(* IEC 61131-3 sources: SIMERLIFT/logiwork_simerlift_80v/logiwork_simerlift_80v/HEMAbattery/src_FBD/fbdCommon, 9 files *)

(* ---- fMaxSint.iecst ---- *)
FUNCTION fMaxSint  {
    width := 200;
  }

VAR_INPUT
	arr:ARRAY[0..15] OF SINT;
	sizeof:USINT;
END_VAR

VAR_OUTPUT
	max : SINT;
END_VAR

VAR
i:USINT;

END_VAR

max:=-128;

FOR i:=1 TO sizeof By 1 DO
	IF max<arr[i-1] THEN
		max:=arr[i-1];
	END_IF;
END_FOR;

END_FUNCTION

(* ---- fMinUint.iecst ---- *)
FUNCTION fMinUint  {
    width := 200;
  }

VAR_INPUT
	arr:ARRAY[0..15] OF UINT;
	sizeof:USINT;
END_VAR

VAR_OUTPUT
	min : UINT;
END_VAR

VAR
i:USINT;

END_VAR

min:=16#FFFF;

FOR i:=1 TO sizeof By 1 DO
	IF min>arr[i-1] THEN
		min:=arr[i-1];
	END_IF;
END_FOR;

END_FUNCTION

(* ---- RBIT.iecfbd ---- *)
FUNCTION RBIT
  VAR_INPUT
    start : INT;
    len : INT;
    INbit : LWORD;
  END_VAR
  VAR_OUTPUT
    OUTbit : LWORD;
  END_VAR

  (*

    // Network 1:
    SHR(IN := INbit, N := start, SHR => @C(12).SHR);
    SUB(IN1 := 64, IN2 := len, SUB => @C(2).SUB);
    SHR(IN := 16#FFFFFFFFFFFFFFFF, N := @C(2).SUB, SHR => @C(6).SHR);
    AND(IN1 := @C(12).SHR, IN2 := @C(6).SHR, AND => OUTbit);

  *)

  @VF(1) : @E(64), @R(460.0, 160.0, 80.0, 19.0), INT;
  @C(2) : @F(SUB), @R(590.0, 160.0, 40.0, 38.0), INT, @I(@N(IN1), @L(9.5)), @I(@N(IN2), @L(29.5)), @O(@N(SUB), @R(9.5));
  @VF(3) : @E(len), @R(230.0, 180.0, 140.0, 19.0);
  @C(6) : @F(SHR), @R(670.0, 140.0, 100.0, 38.0), LWORD, @I(@N(IN), @L(9.5)), @I(@N(N), @L(29.5)), @O(@N(SHR), @R(9.5));
  @VF(8) : @E(16#FFFFFFFFFFFFFFFF), @R(460.0, 140.0, 170.0, 19.0), LWORD;
  @VF(10) : @E(INbit), @R(230.0, 100.0, 140.0, 19.0);
  @VF(11) : @E(start), @R(230.0, 120.0, 140.0, 19.0);
  @C(12) : @F(SHR), @R(670.0, 100.0, 100.0, 38.0), LWORD, @I(@N(IN), @L(9.5)), @I(@N(N), @L(29.5)), @O(@N(SHR), @R(9.5));
  @C(15) : @F(AND), @R(830.0, 100.0, 40.0, 38.0), LWORD, @I(@N(IN1), @L(9.5)), @I(@N(IN2), @L(29.5)), @O(@N(AND), @R(9.5));
  @VF(18) : @E(OUTbit), @R(1000.0, 100.0, 140.0, 19.0);

  @G(4) :
     @L(@VF(3).o, @C(2).IN2)
    ;
  @G(5) :
     @L(@VF(1).o, @C(2).IN1)
    ;
  @G(7) :
     @L(@C(2).SUB, @C(6).N)
    ;
  @G(9) :
     @L(@VF(8).o, @C(6).IN)
    ;
  @G(13) :
     @L(@VF(10).o, @C(12).IN)
    ;
  @G(14) :
     @L(@VF(11).o, @C(12).N)
    ;
  @G(16) :
     @L(@C(12).SHR, @C(15).IN1)
    ;
  @G(17) :
     @L(@C(6).SHR, @C(15).IN2)
    ;
  @G(19) :
     @L(@C(15).AND, @VF(18).i)
    ;
END_FUNCTION

(* ---- WFLT.iecfbd ---- *)
FUNCTION WFLT
  VAR_INPUT
    start : INT;
    len : INT;
    prm : LREAL;
    ofs : LREAL;
    res : LREAL;
  END_VAR
  VAR_OUTPUT
    OUTbit : LWORD;
  END_VAR

  (*

    // Network 1:
    SHL(IN := 16#FFFFFFFFFFFFFFFF, N := start, SHL => @C(4).SHL);
    ADD(IN1 := start, IN2 := len, ADD => @C(7).ADD);
    SUB(IN1 := 64, IN2 := @C(7).ADD, SUB => @C(12).SUB);
    SHR(IN := 16#FFFFFFFFFFFFFFFF, N := @C(12).SUB, SHR => @C(15).SHR);
    AND(IN1 := @C(4).SHL, IN2 := @C(15).SHR, AND => @C(19).AND);
    SUB(IN1 := prm, IN2 := ofs, SUB => @C(29).SUB);
    DIV(IN1 := @C(29).SUB, IN2 := res, DIV => @C(32).DIV);
    TO_LWORD(IN := @C(32).DIV, TO_LWORD => @C(36).TO_LWORD);
    SHL(IN := @C(36).TO_LWORD, N := start, SHL => @C(23).SHL);
    AND(IN1 := @C(19).AND, IN2 := @C(23).SHL, AND => OUTbit);

  *)

  @C(4) : @F(SHL), @R(670.0, 80.0, 100.0, 38.0), LWORD, @I(@N(IN), @L(9.5)), @I(@N(N), @L(29.5)), @O(@N(SHL), @R(9.5));
  @C(12) : @F(SUB), @R(930.0, 100.0, 40.0, 38.0), INT, @I(@N(IN1), @L(9.5)), @I(@N(IN2), @L(29.5)), @O(@N(SUB), @R(9.5));
  @C(15) : @F(SHR), @R(1030.0, 80.0, 100.0, 38.0), LWORD, @I(@N(IN), @L(9.5)), @I(@N(N), @L(29.5)), @O(@N(SHR), @R(9.5));
  @C(19) : @F(AND), @R(1190.0, 60.0, 40.0, 38.0), LWORD, @I(@N(IN1), @L(9.5)), @I(@N(IN2), @L(29.5)), @O(@N(AND), @R(9.5));
  @C(7) : @F(ADD), @R(670.0, 120.0, 40.0, 38.0), INT, @I(@N(IN1), @L(9.5)), @I(@N(IN2), @L(29.5)), @O(@N(ADD), @R(9.5));
  @C(22) : @F(AND), @R(1320.0, 140.0, 40.0, 38.0), LWORD, @I(@N(IN1), @L(9.5)), @I(@N(IN2), @L(29.5)), @O(@N(AND), @R(9.5));
  @C(23) : @F(SHL), @R(670.0, 160.0, 100.0, 38.0), LWORD, @I(@N(IN), @L(9.5)), @I(@N(N), @L(29.5)), @O(@N(SHL), @R(9.5));
  @VF(8) : @E(16#FFFFFFFFFFFFFFFF), @R(470.0, 80.0, 170.0, 19.0), LWORD;
  @VF(1) : @E(start), @R(130.0, 100.0, 140.0, 19.0);
  @VF(11) : @E(64), @R(820.0, 100.0, 70.0, 19.0), INT;
  @VF(17) : @E(16#FFFFFFFFFFFFFFFF), @R(810.0, 80.0, 170.0, 19.0), LWORD;
  @VF(2) : @E(len), @R(130.0, 140.0, 140.0, 19.0);
  @VF(27) : @E(OUTbit), @R(1400.0, 140.0, 140.0, 19.0);
  @VF(3) : @E(prm), @R(130.0, 160.0, 140.0, 19.0);
  @VF(24) : @E(ofs), @R(130.0, 180.0, 140.0, 19.0);
  @C(29) : @F(SUB), @R(320.0, 160.0, 40.0, 38.0), LREAL, @I(@N(IN1), @L(9.5)), @I(@N(IN2), @L(29.5)), @O(@N(SUB), @R(9.5));
  @C(32) : @F(DIV), @R(400.0, 160.0, 40.0, 38.0), LREAL, @I(@N(IN1), @L(9.5)), @I(@N(IN2), @L(29.5)), @O(@N(DIV), @R(9.5));
  @VF(34) : @E(res), @R(130.0, 200.0, 140.0, 19.0);
  @C(36) : @F(TO_LWORD), @R(460.0, 160.0, 120.0, 18.0), LREAL, @I(@N(IN), @L(9.5)), @O(@N(TO_LWORD), @R(9.5));
  @CP(10) : 609.5, 109.5;

  @G(5) :
     @L(@VF(8).o, @C(4).IN)
    ;
  @G(6) :
     @L(@VF(1).o, @CP(10)),
     @L(@CP(10), @C(4).N),
     @L(@CP(10), @C(7).IN1),
     @L(@CP(10), @C(23).N)
    ;
  @G(13) :
     @L(@VF(11).o, @C(12).IN1)
    ;
  @G(14) :
     @L(@C(7).ADD, @C(12).IN2)
    ;
  @G(16) :
     @L(@C(12).SUB, @C(15).N)
    ;
  @G(18) :
     @L(@VF(17).o, @C(15).IN)
    ;
  @G(9) :
     @L(@VF(2).o, @C(7).IN2)
    ;
  @G(20) :
     @L(@C(15).SHR, @C(19).IN2)
    ;
  @G(21) :
     @L(@C(4).SHL, @C(19).IN1)
    ;
  @G(25) :
     @L(@C(19).AND, @C(22).IN1)
    ;
  @G(26) :
     @L(@C(23).SHL, @C(22).IN2)
    ;
  @G(28) :
     @L(@C(22).AND, @VF(27).i)
    ;
  @G(30) :
     @L(@VF(3).o, @C(29).IN1)
    ;
  @G(31) :
     @L(@VF(24).o, @C(29).IN2)
    ;
  @G(33) :
     @L(@C(29).SUB, @C(32).IN1)
    ;
  @G(35) :
     @L(@VF(34).o, @C(32).IN2)
    ;
  @G(37) :
     @L(@C(32).DIV, @C(36).IN)
    ;
  @G(38) :
     @L(@C(36).TO_LWORD, @C(23).IN)
    ;
END_FUNCTION

(* ---- AVG.iecfbd ---- *)
FUNCTION_BLOCK AVG
  {
    In {index := 0};
    Out {index := 0};
    width := 100;
    height := 18;
  }

  VAR
    Out_Buff : LREAL := 0;
  END_VAR
  VAR_INPUT
    In : LREAL := 0;
  END_VAR
  VAR_OUTPUT
    Out : LREAL := 0;
  END_VAR

  (*

    // Network 1:
    MUL(IN1 := In, IN2 := 0.001, MUL => @C(4).MUL);
    MUL(IN1 := Out_Buff, IN2 := 0.999, MUL => @C(9).MUL);
    ADD(IN1 := @C(4).MUL, IN2 := @C(9).MUL, ADD => (Out, Out_Buff));

  *)

  @VF(1) : @E(In), @R(20.0, 20.0, 220.0, 19.0);
  @VF(2) : @E(Out), @R(520.0, 20.0, 220.0, 19.0);
  @VF(186) : @E(0.001), @R(130.0, 40.0, 110.0, 19.0), LREAL;
  @C(6) : @F(ADD), @R(400.0, 20.0, 40.0, 38.0), LREAL, @I(@N(IN1), @L(9.5)), @I(@N(IN2), @L(29.5)), @O(@N(ADD), @R(9.5));
  @VF(10) : @E(0.999), @R(130.0, 80.0, 110.0, 19.0), LREAL;
  @C(4) : @F(MUL), @R(280.0, 20.0, 40.0, 38.0), LREAL, @I(@N(IN1), @L(9.5)), @I(@N(IN2), @L(29.5)), @O(@N(MUL), @R(9.5));
  @C(9) : @F(MUL), @R(280.0, 60.0, 40.0, 38.0), LREAL, @I(@N(IN1), @L(9.5)), @I(@N(IN2), @L(29.5)), @O(@N(MUL), @R(9.5));
  @VF(12) : @E(Out_Buff), @R(520.0, 40.0, 220.0, 19.0);
  @VF(15) : @E(Out_Buff), @R(20.0, 60.0, 220.0, 19.0);
  @CP(13) : 489.5, 29.5;

  @G(14) :
     @L(@C(6).ADD, @CP(13)),
     @L(@CP(13), @VF(2).i),
     @L(@CP(13), @VF(12).i)
    ;
  @G(5) :
     @L(@VF(1).o, @C(4).IN1)
    ;
  @G(8) :
     @L(@VF(186).o, @C(4).IN2)
    ;
  @G(11) :
     @L(@VF(10).o, @C(9).IN2)
    ;
  @G(3) :
     @L(@C(4).MUL, @C(6).IN1)
    ;
  @G(7) :
     @L(@C(9).MUL, @C(6).IN2)
    ;
  @G(16) :
     @L(@VF(15).o, @C(9).IN1)
    ;
END_FUNCTION_BLOCK

(* ---- CounTim.iecfbd ---- *)
FUNCTION_BLOCK CounTim
  {
    ACCper {index := 2};
    DECper {index := 3};
    PV {index := 4};
    CV {index := 4};
    height := 98;
    width := 210;
    bgColor := "darkseagreen";
  }

  VAR
    FLASH7 : FLASH;
    FLASH8 : FLASH;
    CTUD3 : CTUD;
  END_VAR
  VAR_INPUT
    ACCper : TIME;
    DECper : TIME;
    CU : BOOL;
    CD : BOOL;
    PV : INT;
  END_VAR
  VAR_OUTPUT
    CV : INT;
    QU : BOOL;
    QD : BOOL;
  END_VAR

  (*

    // Network 1:
    AND(IN1 := NOT CTUD3.QU, IN2 := CU, AND => @C(66).AND);
    FLASH7(IN := @C(66).AND, PER := ACCper);
    AND(IN1 := CD, IN2 := NOT CTUD3.QD, AND => @C(68).AND);
    FLASH8(IN := @C(68).AND, PER := DECper);
    CTUD3(CU := FLASH7.OUT, CD := FLASH8.OUT, PV := PV, QU => QU, QD => QD, CV => CV);

  *)

  @C(66) : @F(AND), @R(410.0, 240.0, 40.0, 38.0), BOOL, @I(@N(IN1), @L(9.5), @NEG), @I(@N(IN2), @L(29.5)), @O(@N(AND), @R(9.5));
  @C(39) : @FB(FLASH7), @R(550.0, 260.0, 120.0, 38.0), @I(@N(IN), @L(9.5)), @I(@N(PER), @L(29.5)), @O(@N(OUT), @R(9.5));
  @C(40) : @FB(FLASH8), @R(550.0, 300.0, 120.0, 38.0), @I(@N(IN), @L(9.5)), @I(@N(PER), @L(29.5)), @O(@N(OUT), @R(9.5));
  @C(41) : @FB(CTUD3), @R(780.0, 260.0, 100.0, 98.0), @I(@N(CU), @L(9.5)), @I(@N(CD), @L(29.5)), @I(@N(R), @L(49.5)), @I(@N(LD), @L(69.5)), @I(@N(PV), @L(89.5)), @O(@N(QU), @R(9.5)), @O(@N(QD), @R(29.5)), @O(@N(CV), @R(89.5));
  @C(68) : @F(AND), @R(410.0, 340.0, 40.0, 38.0), BOOL, @I(@N(IN1), @L(9.5)), @I(@N(IN2), @L(29.5), @NEG), @O(@N(AND), @R(9.5));
  @VF(1) : @E(CU), @R(120.0, 260.0, 140.0, 19.0);
  @VF(3) : @E(ACCper), @R(120.0, 280.0, 140.0, 19.0);
  @VF(6) : @E(DECper), @R(120.0, 320.0, 140.0, 19.0);
  @VF(8) : @E(CD), @R(120.0, 340.0, 140.0, 19.0);
  @VF(10) : @E(PV), @R(120.0, 390.0, 140.0, 19.0);
  @VF(12) : @E(CV), @R(980.0, 340.0, 140.0, 19.0);
  @VF(14) : @E(QD), @R(980.0, 280.0, 140.0, 19.0);
  @VF(15) : @E(QU), @R(980.0, 260.0, 140.0, 19.0);
  @CP(17) : 929.5, 269.5;
  @CP(18) : 929.5, 289.5;

  @G(67) :
     @L(@C(66).AND, @C(39).IN)
    ;
  @G(46) :
     @L(@C(39).OUT, @C(41).CU)
    ;
  @G(47) :
     @L(@C(40).OUT, @C(41).CD)
    ;
  @G(69) :
     @L(@C(68).AND, @C(40).IN)
    ;
  @G(2) :
     @L(@VF(1).o, @C(66).IN2)
    ;
  @G(4) :
     @L(@VF(3).o, @C(39).PER)
    ;
  @G(7) :
     @L(@VF(6).o, @C(40).PER)
    ;
  @G(9) :
     @L(@VF(8).o, @C(68).IN1)
    ;
  @G(11) :
     @L(@VF(10).o, @C(41).PV)
    ;
  @G(13) :
     @L(@C(41).CV, @VF(12).i)
    ;
  @G(5) :
     @L(@C(41).QD, @CP(18)),
     @L(@CP(18), @VF(14).i),
     @L(@CP(18), @C(68).IN2)
    ;
  @G(16) :
     @L(@C(41).QU, @CP(17)),
     @L(@CP(17), @VF(15).i),
     @L(@CP(17), @C(66).IN1)
    ;
END_FUNCTION_BLOCK

(* ---- FLASH.iecfbd ---- *)
FUNCTION_BLOCK FLASH
  VAR
    TON2 : TON;
    TON1 : TON;
  END_VAR
  VAR_INPUT
    IN : BOOL := 0;
    PER : TIME := T#0s;
  END_VAR
  VAR_OUTPUT
    OUT : BOOL := 0;
  END_VAR

  (*

    // Network 1:
    TON2(IN := TON1.Q, PT := PER);
    NOT(IN := TON2.Q, NOT => @C(5).NOT);
    AND(IN1 := IN, IN2 := @C(5).NOT, AND => @C(4).AND);
    TON1(IN := @C(4).AND, PT := PER, Q => OUT);

  *)

  @C(2) : @FB(TON2), @R(910.0, 290.0, 100.0, 38.0), @I(@N(IN), @L(9.5)), @I(@N(PT), @L(29.5)), @O(@N(Q), @R(9.5)), @O(@N(ET), @R(29.5));
  @C(5) : @F(NOT), @R(450.0, 190.0, 60.0, 18.0), BOOL, @I(@N(IN), @L(9.5)), @O(@N(NOT), @R(9.5));
  @C(1) : @FB(TON1), @R(730.0, 170.0, 100.0, 38.0), @I(@N(IN), @L(9.5)), @I(@N(PT), @L(29.5)), @O(@N(Q), @R(9.5)), @O(@N(ET), @R(29.5));
  @C(4) : @F(AND), @R(570.0, 170.0, 40.0, 38.0), BOOL, @I(@N(IN1), @L(9.5)), @I(@N(IN2), @L(29.5)), @O(@N(AND), @R(9.5));
  @VF(11) : @E(OUT), @R(990.0, 170.0, 140.0, 19.0);
  @VF(9) : @E(IN), @R(290.0, 170.0, 140.0, 19.0);
  @VF(13) : @E(PER), @R(260.0, 310.0, 140.0, 19.0);
  @CP(15) : 669.5, 319.5;
  @CP(12) : 869.5, 179.5;

  @G(14) :
     @L(@VF(13).o, @CP(15)),
     @L(@CP(15), @C(1).PT),
     @L(@CP(15), @C(2).PT)
    ;
  @G(6) :
     @L(@C(5).NOT, @C(4).IN2)
    ;
  @G(7) :
     @L(@C(2).Q, @C(5).IN)
    ;
  @G(3) :
     @L(@C(1).Q, @CP(12)),
     @L(@CP(12), @C(2).IN),
     @L(@CP(12), @VF(11).i)
    ;
  @G(8) :
     @L(@C(4).AND, @C(1).IN)
    ;
  @G(10) :
     @L(@VF(9).o, @C(4).IN1)
    ;
END_FUNCTION_BLOCK

(* ---- Mosfet_BTTdiag.iecst ---- *)
FUNCTION_BLOCK  BTTdiag  {  width := 200;   }

VAR_INPUT
	IN   : BOOL;
	Iout : UINT;
	Imin : UINT;
	Imax : UINT;
END_VAR

VAR_OUTPUT
	DIAG :BYTE;
		/*DIN_DIAG
		 * 0: no problem
		 * 01: under current / no load
		 * 02: over current
		 * 03: chip error*/
END_VAR

DIAG:=0;

IF IN THEN
	IF Iout<Imin THEN
		DIAG:=1;
	ELSIF Iout>Imax THEN
		DIAG:=2;
	END_IF;
ELSIF Iout>Imin THEN
	DIAG:=3;
END_IF;
END_FUNCTION_BLOCK

(* ---- Tbuffer.iecfbd ---- *)
FUNCTION_BLOCK Tbuffer
  {
    bgColor := "darkgray";
  }

  VAR
    TOF1 : TOF;
    TON1 : TON;
  END_VAR
  VAR_INPUT
    I : BOOL := 0;
    D : TIME;
  END_VAR
  VAR_OUTPUT
    O : BOOL := 0;
  END_VAR

  (*

    // Network 1:
    TON1(IN := I, PT := D);
    TOF1(IN := TON1.Q, PT := D, Q => O);

  *)

  @C(3) : @FB(TOF1), @R(650.0, 60.0, 100.0, 38.0), @I(@N(IN), @L(9.5)), @I(@N(PT), @L(29.5)), @O(@N(Q), @R(9.5)), @O(@N(ET), @R(29.5));
  @C(4) : @FB(TON1), @R(470.0, 60.0, 100.0, 38.0), @I(@N(IN), @L(9.5)), @I(@N(PT), @L(29.5)), @O(@N(Q), @R(9.5)), @O(@N(ET), @R(29.5));
  @VF(2) : @E(O), @R(790.0, 60.0, 220.0, 19.0);
  @VF(1) : @E(I), @R(170.0, 60.0, 220.0, 19.0);
  @VF(11) : @E(D), @R(200.0, 100.0, 140.0, 19.0);
  @CP(9) : 429.5, 109.5;

  @G(7) :
     @L(@C(3).Q, @VF(2).i)
    ;
  @G(6) :
     @L(@C(4).Q, @C(3).IN)
    ;
  @G(5) :
     @L(@VF(1).o, @C(4).IN)
    ;
  @G(8) :
     @L(@CP(9), @C(3).PT),
     @L(@CP(9), @C(4).PT),
     @L(@VF(11).o, @CP(9))
    ;
END_FUNCTION_BLOCK
